FUNCTION_BLOCK SxDuo
VAR_INPUT
	EN: BOOL;
	FireAlarm: BOOL;
	Damper1Alarm: BOOL;
	Exercising: BOOL;
	Damper2Alarm: BOOL;
	Damper1Open: BOOL;
	Damper1Closed: BOOL;
	Damper2Open: BOOL;
	Damper2Closed: BOOL;
	ServiceAlarm: BOOL;
END_VAR
VAR_OUTPUT
	ENO: BOOL;
	FireAlarmOut: bool;
	ActivateFireAlarm: BOOL;
	ResetSmokeDetector: BOOL;
	ForceExercise: BOOL;
END_VAR
VAR
END_VAR

ENO := EN;
IF EN THEN
	FireAlarmOut := FireAlarm;	
END_IF

END_FUNCTION_BLOCK

(* stored: Version 1.1.0.1, ProductVersion 3.1.4024.4
   POU SxDuo: Id {4cb84e5e-c02e-41d2-853c-6427b6e8aeeb}, SpecialFunc None *)
